TYPE ST_TD400Control :  (* Serial communication defined in Oerlikon Leybold Manual GA05281_002_C0 *)
STRUCT
    {attribute 'pytmc' := '
    pv: SetPumpSpeed;
    io: i;
    '}
    wSetSetpointFreq_P24: WORD; // speed setting in Hz
END_STRUCT
END_TYPE

(* stored: Version 1.1.0.1
   DUT ST_TD400Control: Id {1be82e89-db71-431e-815d-0070384e019c} *)
